// TIA Portal V17 export
// export: Created 2022-12-09T10:50:29.1584279Z, ExportSetting WithDefaults, DisplayName Totally Integrated Automation Portal, DisplayVersion V17 Update 5, DisplayName TIA Portal Openness, DisplayVersion V17 Update 5, DisplayName TIA Portal Version Control Interface, DisplayVersion V17, DisplayName Simotion SCOUT TIA, DisplayVersion 5.4.3.0, DisplayName SINAMICS Startdrive Advanced, DisplayVersion V17 SP1, DisplayName SINAMICS Startdrive G130, G150, S120, S150, SINAMICS MV, S210, DisplayVersion V17 SP1, DisplayName SINAMICS Startdrive G110M, G120, G120C, G120D, G120P, G115D, DisplayVersion V17 SP1, DisplayName STEP 7 Professional, DisplayVersion V17 Update 5, DisplayName STEP 7 Safety, DisplayVersion V17, DisplayName WinCC Advanced, DisplayVersion V17 Update 5
VAR_GLOBAL   // PLC tag table "OMAC_Constants"
END_VAR
VAR_GLOBAL CONSTANT   // user constants
   OMAC_MODE_INVALID : DInt := 0;
   OMAC_MODE_PRODUCTION : DInt := 1;
   OMAC_MODE_MANUAL : DInt := 3;
   OMAC_MODE_MAINTENANCE : DInt := 2;
   OMAC_MODE_CHANGE_OVER : DInt := 4;
   OMAC_MODE_CLEAN : DInt := 5;
   OMAC_MODE_SET_UP : DInt := 6;
   OMAC_MODE_EMPTY_OUT : DInt := 7;
   OMAC_MODE_OEM_SPECIFIC : DInt := 8;
   OMAC_MODE_USER_01 : DInt := 10;
   OMAC_MODE_USER_02 : DInt := 11;
   OMAC_MODE_USER_03 : DInt := 12;
   OMAC_MODE_USER_04 : DInt := 13;
   OMAC_MODE_USER_05 : DInt := 14;
   OMAC_STATE_UNDEFINED : DInt := 0;
   OMAC_STATE_CLEARING : DInt := 1;
   OMAC_STATE_STOPPED : DInt := 2;
   OMAC_STATE_STARTING : DInt := 3;
   OMAC_STATE_IDLE : DInt := 4;
   OMAC_STATE_SUSPENDED : DInt := 5;
   OMAC_STATE_EXECUTE : DInt := 6;
   OMAC_STATE_STOPPING : DInt := 7;
   OMAC_STATE_ABORTING : DInt := 8;
   OMAC_STATE_ABORTED : DInt := 9;
   OMAC_STATE_HOLDING : DInt := 10;
   OMAC_STATE_HELD : DInt := 11;
   OMAC_STATE_UNHOLDING : DInt := 12;
   OMAC_STATE_SUSPENDING : DInt := 13;
   OMAC_STATE_UNSUSPENDING : DInt := 14;
   OMAC_STATE_RESETTING : DInt := 15;
   OMAC_STATE_COMPLETING : DInt := 16;
   OMAC_STATE_COMPLETE : DInt := 17;
   OMAC_CMD_UNDEFINED : DInt := 0;
   OMAC_CMD_RESET : DInt := 1;
   OMAC_CMD_START : DInt := 2;
   OMAC_CMD_STOP : DInt := 3;
   OMAC_CMD_HOLD : DInt := 4;
   OMAC_CMD_UNHOLD : DInt := 5;
   OMAC_CMD_SUSPEND : DInt := 6;
   OMAC_CMD_UNSUSPEND : DInt := 7;
   OMAC_CMD_ABORT : DInt := 8;
   OMAC_CMD_CLEAR : DInt := 9;
   OMAC_CMD_COMPLETE : DInt := 10;
   OMAC_LANGUAGE_1 : Int := 0;
   OMAC_LANGUAGE_2 : Int := 1;
   OMAC_DIAG_BUFFER_UPPER_LIM : Int := 15;
   OMAC_LANGUAGES_UPPER_LIM : Int := 1;
   OMAC_MODES_UPPER_LIM : Int := 14;
   OMAC_STATES_UPPER_LIM : Int := 17;
   OMAC_MAX_MODES_UPPER_LIM : Int := 14;
   OMAC_MODE_SPARE : DInt := 9;
   UPPEROMACMODE : Int := 31;
END_VAR
